FUNCTION_BLOCK ST_AND
  (* Standard: 61499-1-D.1; Classification: Boolean functions *)
  (* Version 0.1, 2001-08-05, JHC, Rockwell Automation, XML version *)
  (* Version 0.0, 1999-02-20, JHC, Rockwell Automation, SRC version *)
  (* Compiler header: package fb.rt.math; *)
  (* Compiler classdef: class FB_AND extends FBFunction2 *)
  (* Compiler Java IBM VisualAge 3.0 *)
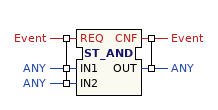
  EVENT_INPUT
    REQ WITH IN1, IN2;
  END_EVENT
  EVENT_OUTPUT
    CNF WITH OUT;
  END_EVENT
  VAR_INPUT
    IN1 : ANY;
    IN2 : ANY;
  END_VAR
  VAR_OUTPUT
    OUT : ANY; (* Result *)
  END_VAR
  ALGORITHM REQ IN JAVA:

  END_ALGORITHM
END_FUNCTION_BLOCK
